(* IEC 61131-3 sources: IRIS-Project/LASAL CONTROL SOFTWARE/LasalProject_2025_09_12/Class/ClasseEsempiotimer, 1 file *)

(* ---- ClasseEsempiotimer.st ---- *)
(*!
<Class
	Name               = "ClasseEsempiotimer"
	Revision           = "0.0"
	RealtimeTask       = "true"
	CyclicTask         = "true"
	DefCyclictime      = "100 ms"
	BackgroundTask     = "false"
	Sigmatek           = "false"
	OSInterface        = "false"
	HighPriority       = "false"
	Automatic          = "false"
	UpdateMode         = "Prescan"
	SharedCommandTable = "true"
	Objectsize         = "(284,120)">
	<Channels>
		<Server Name="ClassSvr" Visualized="false" Initialize="false" WriteProtected="true" Retentive="false"/>
		<Client Name="Client" Required="true" Internal="false"/>
	</Channels>
</Class>
*)
ClasseEsempiotimer : CLASS
  //Servers:
	ClassSvr 	: SvrChCmd_DINT;
  //Clients:
	Client 	: CltChCmd_TimerLib;
  //Variables:
		Variable 	: DINT;
		pointertime 	: ^UDINT;
		v_timer 	: UDINT;
		c_timer 	: DINT;
		ActTimer 	: UDINT;
		Timerremain 	: UDINT;
		A 	: DINT;
  //Functions:

	FUNCTION VIRTUAL GLOBAL Init;

	FUNCTION VIRTUAL GLOBAL CyWork
		VAR_INPUT
			EAX 	: UDINT;
		END_VAR
		VAR_OUTPUT
			state (EAX) 	: UDINT;
		END_VAR;

	FUNCTION VIRTUAL GLOBAL RtWork
		VAR_INPUT
			EAX 	: UDINT;
		END_VAR
		VAR_OUTPUT
			state (EAX) 	: UDINT;
		END_VAR;
  //Tables:
	FUNCTION @STD
		VAR_OUTPUT
			ret_code	: CONFSTATES;
		END_VAR;
	FUNCTION GLOBAL TAB @CT_;
END_CLASS;

#pragma usingLtd TimerLib

FUNCTION VIRTUAL GLOBAL ClasseEsempiotimer::RtWork
	VAR_INPUT
		EAX 	: UDINT;
	END_VAR
	VAR_OUTPUT
		state (EAX) 	: UDINT;
	END_VAR

	state := READY;

END_FUNCTION

FUNCTION VIRTUAL GLOBAL ClasseEsempiotimer::CyWork
	VAR_INPUT
		EAX 	: UDINT;
	END_VAR
	VAR_OUTPUT
		state (EAX) 	: UDINT;
	END_VAR

  case c_timer of

    0:
    Client.TimerStart(pudStartTime:=#v_timer);
    c_timer:=1;

    1:
      if Client.IsTimerFinished(pudStartTime:=#v_timer, udDuration:=50000) then
        c_timer:=2;
      end_if;

      ActTimer:=Client.TimerAct(pudStartTime:=#v_timer);
      Timerremain:=Client.TimerRest(pudStartTime:=#v_timer, udDuration:=50000);

  end_case;

	state := READY;

END_FUNCTION

FUNCTION VIRTUAL GLOBAL ClasseEsempiotimer::Init
Variable:=0;
v_timer:=0;
pointertime:=#v_timer;
c_timer:=0;
ActTimer:=0;
Timerremain:=0;
A:=0;
END_FUNCTION
